// TIA Portal V17 export
// export: Created 2023-03-06T02:05:14.6927948Z, ExportSetting WithDefaults, DisplayName Totally Integrated Automation Portal, DisplayVersion V17 Update 4, DisplayName TIA Portal Openness, DisplayVersion V17 Update 4, DisplayName TIA Portal Version Control Interface, DisplayVersion V17, DisplayName STEP 7 Professional, DisplayVersion V17 Update 4, DisplayName STEP 7 Safety, DisplayVersion V17, DisplayName WinCC Professional, DisplayVersion V17 Update 4
DATA_BLOCK "PCS1"   // DB41
{ S7_Optimized_Access := 'TRUE' }
VERSION : 0.1
// stored: AutoNumber false, DBAccessibleFromOPCUA true, DBAccessibleFromWebserver true, IsOnlyStoredInLoadMemory false, IsRetainMemResEnabled false, IsWriteProtectedInAS false, MemoryReserve 100
   VAR RETAIN
      TCON { S7_SetPoint := 'True'} : TCON_IP_v4;
   END_VAR
   VAR
      arrData : Array[1..125] of Word;
      xREQ : Bool;
      iCountDone : Int := 1;
      iCountRead : Int := 1;
      MBmode : USInt;
      MBdataAddr : UDInt;
      MBdataLen : UInt;
   END_VAR
   VAR RETAIN
      TCON10 { S7_SetPoint := 'True'} : TCON_IP_v4;
   END_VAR
   VAR
      arrData10 : Array[1..125] of Word;
      xREQ10 : Bool;
      iCountDone10 : Int := 1;
      iCountRead10 : Int := 1;
      MBmode10 : USInt;
      MBdataAddr10 : UDInt;
      MBdataLen10 : UInt;
      R { S7_SetPoint := 'True'} : "R_PE";
      RW { S7_SetPoint := 'True'} : "RW_PE";
      W { S7_SetPoint := 'True'} : "W_PE";
   END_VAR
   VAR RETAIN
      TCONW { S7_SetPoint := 'True'} : TCON_IP_v4;
   END_VAR
   VAR
      arrDataW : Array[1..125] of Word;
      xREQW : Bool;
      iCountDoneW : Int := 1;
      iCountReadW : Int := 1;
      MBmodeW : USInt;
      MBdataAddrW : UDInt;
      MBdataLenW : UInt;
      xDCbus1Avl : Bool;
      xDCbus2Avl : Bool;
      xLVRT : Bool;
      xOVRT : Bool;
      xCommFltSt : Bool;
      xFltSt : Bool;
      xWarnSt : Bool;
      xModFltBus1St : Bool;
      xModFltBus2St : Bool;
      xMod1FltSt : Bool;
      xMod2FltSt : Bool;
      xMod3FltSt : Bool;
      xMod4FltSt : Bool;
      xMod5FltSt : Bool;
      xMod6FltSt : Bool;
      xMod1WarnSt : Bool;
      xMod2WarnSt : Bool;
      xMod3WarnSt : Bool;
      xMod4WarnSt : Bool;
      xMod5WarnSt : Bool;
      xMod6WarnSt : Bool;
      rMod1MaxTemp : Real;
      rMod2MaxTemp : Real;
      rMod3MaxTemp : Real;
      rMod4MaxTemp : Real;
      rMod5MaxTemp : Real;
      rMod6MaxTemp : Real;
      rPacBus1Meas : Real;
      rPacBus2Meas : Real;
      rQacBus1Meas : Real;
      rQacBus2Meas : Real;
      rVacMeas : Real;
      rIacTotMeas : Real;
      iCodeFlt : Int;
      iCodeWarn : Int;
      iModFlt : Int;
      iModWarn : Int;
      wInvFlt1 : Word;
      wInvFlt2 : Word;
      wInvFlt3 : Word;
      wInvFlt4 : Word;
      wInvFlt5 : Word;
      wInvFlt6 : Word;
      wInvFlt7 : Word;
      wInvWarn1 : Word;
      wInvWarn2 : Word;
      wInvWarn3 : Word;
      wInvWarn4 : Word;
      wInvWarn5 : Word;
      wInvWarn6 : Word;
      wMod1Flt1 : Word;
      wMod1Flt2 : Word;
      wMod1Flt3 : Word;
      wMod1Flt4 : Word;
      wMod2Flt1 : Word;
      wMod2Flt2 : Word;
      wMod2Flt3 : Word;
      wMod2Flt4 : Word;
      wMod3Flt1 : Word;
      wMod3Flt2 : Word;
      wMod3Flt3 : Word;
      wMod3Flt4 : Word;
      wMod4Flt1 : Word;
      wMod4Flt2 : Word;
      wMod4Flt3 : Word;
      wMod4Flt4 : Word;
      wMod5Flt1 : Word;
      wMod5Flt2 : Word;
      wMod5Flt3 : Word;
      wMod5Flt4 : Word;
      wMod6Flt1 : Word;
      wMod6Flt2 : Word;
      wMod6Flt3 : Word;
      wMod6Flt4 : Word;
      wMod1Warn1 : Word;
      wMod1Warn2 : Word;
      wMod1Warn3 : Word;
      wMod1Warn4 : Word;
      wMod2Warn1 : Word;
      wMod2Warn2 : Word;
      wMod2Warn3 : Word;
      wMod2Warn4 : Word;
      wMod3Warn1 : Word;
      wMod3Warn2 : Word;
      wMod3Warn3 : Word;
      wMod3Warn4 : Word;
      wMod4Warn1 : Word;
      wMod4Warn2 : Word;
      wMod4Warn3 : Word;
      wMod4Warn4 : Word;
      wMod5Warn1 : Word;
      wMod5Warn2 : Word;
      wMod5Warn3 : Word;
      wMod5Warn4 : Word;
      wMod6Warn1 : Word;
      wMod6Warn2 : Word;
      wMod6Warn3 : Word;
      wMod6Warn4 : Word;
      aWbit : Struct
         xStart : Word;
         xStopW : Word;
         xResetW : Word;
         xEnableW : Word;
         xEmergency : Word;
      END_STRUCT;
   END_VAR
BEGIN
   TCON.RemoteAddress.ADDR[1] := 192;
   TCON.RemoteAddress.ADDR[2] := 168;
   TCON.RemoteAddress.ADDR[3] := 150;
   TCON.RemoteAddress.ADDR[4] := 44;
   TCON10.RemoteAddress.ADDR[1] := 192;
   TCON10.RemoteAddress.ADDR[2] := 168;
   TCON10.RemoteAddress.ADDR[3] := 150;
   TCON10.RemoteAddress.ADDR[4] := 44;
   TCONW.RemoteAddress.ADDR[1] := 192;
   TCONW.RemoteAddress.ADDR[2] := 168;
   TCONW.RemoteAddress.ADDR[3] := 150;
   TCONW.RemoteAddress.ADDR[4] := 44;
END_DATA_BLOCK
